(* IEC 61131-3 sources: Industry-PLC-LLM/data/PLCBEAD_repo/PLCBEAD_PLCEmbed-main/PLC-BEAD/Source/GEB/SDT_TO_DT, 1 file *)

(* ---- SDT_TO_DT.ST ---- *)
TYPE oscat_SDT :
	STRUCT
		YEAR  : INT;
		MONTH : INT;
		DAY  : INT;
		WEEKDAY  : INT;
		HOUR : INT;
		MINUTE : INT;
		SECOND : INT;
		MS : INT;
	END_STRUCT;
END_TYPE

FUNCTION _INT_TO_UDINT:UDINT
	VAR_INPUT
		IN :	INT;
	END_VAR

	_INT_TO_UDINT := DINT_TO_UDINT(INT_TO_DINT(IN));
END_FUNCTION

FUNCTION SET_DATE:UDINT

	VAR_INPUT
		YEAR  :	INT;
		MONTH :	INT;
		DAY  :	INT;
	END_VAR

	VAR
		count :	INT;
	END_VAR

	IF MONTH > 2 THEN
		count := (MONTH - 1) * 30;
		IF MONTH > 7 THEN
			count := count + DWORD_TO_INT(SHR(DINT_TO_DWORD(INT_TO_DINT(MONTH) - INT_TO_DINT(3)),1));
		ELSE
			count := count + DWORD_TO_INT(SHR(DINT_TO_DWORD(INT_TO_DINT(MONTH) - INT_TO_DINT(4)),1));
		END_IF;
		IF SHL(INT_TO_WORD(YEAR),14) = WORD#0 THEN
			count := count + 1;
		END_IF;
	ELSE
		count := (MONTH - 1) * 31;
	END_IF;
	SET_DATE := (_INT_TO_UDINT(count + DAY  - 1) + DWORD_TO_UDINT(SHR(UDINT_TO_DWORD(_INT_TO_UDINT(YEAR) * UDINT#1461 - UDINT#2878169), 2))) * UDINT#86400;

END_FUNCTION

FUNCTION SET_DT:UDINT
	VAR_INPUT
		YEAR  :	INT;
		MONTH :	INT;
		DAY  :	INT;
		HOUR :	INT;
		MINUTE :	INT;
		SECOND :	INT;
	END_VAR

	SET_DT := SET_DATE(YEAR, MONTH, DAY) + _INT_TO_UDINT(SECOND) + _INT_TO_UDINT(MINUTE) * UDINT#60 + _INT_TO_UDINT(HOUR) * UDINT#3600;
END_FUNCTION

FUNCTION_BLOCK SDT_TO_DT_Block

	VAR_INPUT
		DTI :	oscat_SDT;
	END_VAR

	VAR_OUTPUT
		SDT_TO_DT :	UDINT;
	END_VAR

	SDT_TO_DT := SET_DT(DTI.YEAR, DTI.MONTH, DTI.DAY, DTI.HOUR, DTI.MINUTE, DTI.SECOND);

END_FUNCTION_BLOCK

PROGRAM program0

	VAR
		DTI :	oscat_SDT;
		SDT_TO_DT :	UDINT;
		func_block : SDT_TO_DT_Block;
  	END_VAR
	func_block.DTI  :=	DTI;
	func_block();
	SDT_TO_DT := func_block.SDT_TO_DT;

END_PROGRAM
